// Mitsubishi GX Works2 project: 240430_timechart07_직병렬회로   PLC: Q03UDV

PROGRAM MAIN
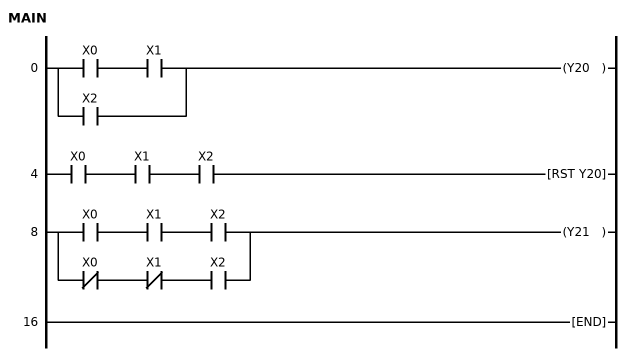
0     LD      X0
      AND     X1
      OR      X2
      OUT     Y20
4     LD      X0
      AND     X1
      AND     X2
      RST     Y20
8     LD      X0
      AND     X1
      AND     X2
      LDI     X0
      ANI     X1
      AND     X2
      ORB
      OUT     Y21
16    END
END_PROGRAM
